% RSLogix 500 project PROC1_COMPARATORS_BAK004.RSS, saved by version 8.30.00.16 %
PROJECT "PROC1"    % processor: Bul.1763 MicroLogix 1100 Series B %

PROGRAM FILES
  LAD 2 "MAIN"  2 rungs
  LAD 3 "COMPARATOR"  9 rungs

DATA FILES
  O0 OUTPUT  4 elements
  I1 INPUT  6 elements
  S2 STATUS  66 elements
  B3 BINARY  1 elements
  T4 TIMER  1 elements
  C5 COUNTER  1 elements
  R6 CONTROL  1 elements
  N7 INTEGER  1 elements
  F8 FLOAT  1 elements

LADDER 2 "MAIN"
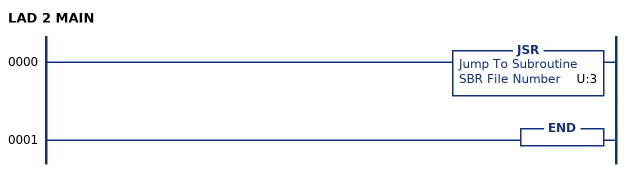
% Rung: 0 %  % edit flag set %
SOR JSR U:3 EOR
% Rung: 1 %
SOR END EOR

LADDER 3 "COMPARATOR"
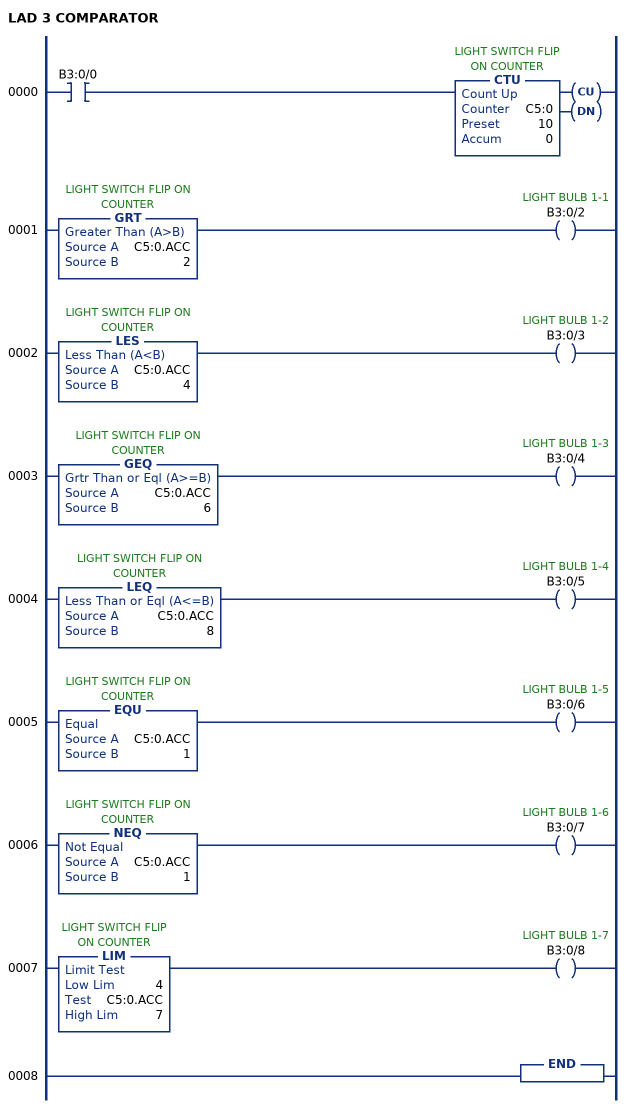
% Rung: 0 %
SOR XIC B3:0/0 CTU C5:0 10 0 EOR
%   C5:0  "LIGHT SWITCH FLIP ON COUNTER" %
% Rung: 1 %
SOR GRT C5:0.ACC 2 OTE B3:0/2 EOR
%   C5:0  "LIGHT SWITCH FLIP ON COUNTER" %
%   B3:0/2  "LIGHT BULB 1-1" %
% Rung: 2 %
SOR LES C5:0.ACC 4 OTE B3:0/3 EOR
%   C5:0  "LIGHT SWITCH FLIP ON COUNTER" %
%   B3:0/3  "LIGHT BULB 1-2" %
% Rung: 3 %
SOR GEQ C5:0.ACC 6 OTE B3:0/4 EOR
%   C5:0  "LIGHT SWITCH FLIP ON COUNTER" %
%   B3:0/4  "LIGHT BULB 1-3" %
% Rung: 4 %
SOR LEQ C5:0.ACC 8 OTE B3:0/5 EOR
%   C5:0  "LIGHT SWITCH FLIP ON COUNTER" %
%   B3:0/5  "LIGHT BULB 1-4" %
% Rung: 5 %
SOR EQU C5:0.ACC 1 OTE B3:0/6 EOR
%   C5:0  "LIGHT SWITCH FLIP ON COUNTER" %
%   B3:0/6  "LIGHT BULB 1-5" %
% Rung: 6 %
SOR NEQ C5:0.ACC 1 OTE B3:0/7 EOR
%   C5:0  "LIGHT SWITCH FLIP ON COUNTER" %
%   B3:0/7  "LIGHT BULB 1-6" %
% Rung: 7 %
SOR LIM 4 C5:0.ACC 7 OTE B3:0/8 EOR
%   C5:0  "LIGHT SWITCH FLIP ON COUNTER" %
%   B3:0/8  "LIGHT BULB 1-7" %
% Rung: 8 %
SOR END EOR

OTHER DOCUMENTED ADDRESSES
  B3:0  "LIGHT SWITCH 1"

REVISION NOTES
  0: Initial code
  1: Added JSR

DATA TABLE (non-zero values as saved)
DATA C5
% .PRE .ACC %
% C5:0 % 10 0
